FUNCTION_BLOCK cross_product (* Basic FB with empty ECC *)
  (* Standard: 61499-2 *)
  (* Version 1.0, 2021-04-13, Lenovo *)
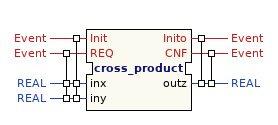
  EVENT_INPUT
    Init WITH inx, iny;
    REQ WITH inx, iny;
  END_EVENT
  EVENT_OUTPUT
    Inito WITH outz;
    CNF WITH outz;
  END_EVENT
  VAR_INPUT
    inx : REAL;
    iny : REAL;
  END_VAR
  VAR_OUTPUT
    outz : REAL;
  END_VAR
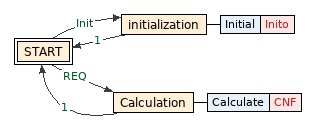
  EC_STATES
    START; (* Initial State *)
    initialization : Initial -> Inito;
    Calculation : Calculate -> CNF;
  END_STATES
  EC_TRANSITIONS
    START TO initialization := Init;
    initialization TO START := 1;
    START TO Calculation := REQ;
    Calculation TO START := 1;
  END_TRANSITIONS
  ALGORITHM Initial IN ST: (* New Algorithm *)

  END_ALGORITHM
  ALGORITHM Calculate IN ST: (* New Algorithm *)
outz:=inx*iny;
  END_ALGORITHM
END_FUNCTION_BLOCK
